// Short string.
// Size is a parameter located at FSParam_Core.nFST_SSTR_SIZE. | DEFAULT: 40
TYPE FsT_SStr : STRING(FSParam_Core.SSTR_SIZE); END_TYPE

(* stored: Version 1.1.0.1, ProductVersion 3.1.4024.4
   DUT FsT_SStr: Id {d9a41d8b-203e-4847-bd7b-75d6c9ced2a1} *)
